FUNCTION_BLOCK "FbTON"
TITLE = 'Таймер с задержкой на включение.'

{ S7_read_back := 'true' ;
  S7_blockview := 'big'  }

AUTHOR  : VA
FAMILY  : LIB_PLC
VERSION : '2.2'

VAR_INPUT // Входные переменные, сохраняемые.
In          :BOOL := FALSE; // Вход таймера.
TimeDelayOn :DINT := 5000 ; // Время задержки включения [мс].
Ts_ms       :DINT := 100  ; // Шаг дискретизации по времени [мс].
END_VAR

VAR_OUTPUT // Выходные переменные, сохраняемые.
Out :BOOL := FALSE; // Выход таймера.
END_VAR

VAR // Внутренние переменные, сохраняемые.
Timer1 :DINT := 0; // Текущее время таймер1 [мс].
END_VAR

BEGIN

// Таймер с задержкой на включение.
//          DbTON
//    +----------------+
//    |     FbTON      |
// ->-|In           Out|->-
//   -|TimeDelayOn     |
//   -|Ts_ms           |
//    +----------------+

IF (TimeDelayOn > 0) THEN // Таймер включен.
  IF (In) THEN // На входе 1.
    IF (Out) THEN // На выходе 1.
    Out := TRUE;
    Timer1 := 0;
    ELSE // На выходе 0.
      IF (Timer1 >= TimeDelayOn) THEN // Задержка включения закончилась.
      Out := TRUE;
      Timer1 := 0;
      ELSE // Задержка включения активна.
      Out := FALSE;
      Timer1 := Timer1 + Ts_ms;
      END_IF;
    END_IF;
  ELSE // Если на входе 0 то на выходе тоже 0.
  Out := FALSE;
  Timer1 := 0;
  END_IF;
ELSE // Таймер выключен.
Out := In;
Timer1 := 0;
END_IF;

// Применение.
//
// При поступлении входного сигнала выходной сигнал появляется не сразу, а с задержкой TimeDelayOn.
// Блок может применятся как фильтр дребезга контактов дискретных входов.
// Совместно с инвертором может применяться для генерации импульсов.

// Временная характеристика.
//
//  In
//  ^
//  | TimeDelayOn           TimeDelayOn
//  |   |<--->|               |<--->|
// 1|   ***********     * *   ***********
//  |   *         *     * *   *         *
// 0*****---------*************---------*****----> t[s]
//
//  Out
//  ^
//  | TimeDelayOn           TimeDelayOn
//  |   |<--->|               |<--->|
// 1|   |     *****           |     *****
//  |   |     *   *           |     *   *
// 0***********---*******************---*****----> t[s]

// @COPYLEFT ALL WRONGS RESERVED :)
// Author: VA
// Contacts: DIY.PLC.314@gmail.com
// Date start LIB_PLC: 2014
// License: GNU GPL-2.0-or-later
// https://www.gnu.org/licenses/old-licenses/gpl-2.0.html
// https://www.youtube.com/watch?v=n1F_MfLRlX0
// https://www.youtube.com/@DIY_PLC
// https://github.com/DIYPLC/LIB_PLC
// https://oshwlab.com/diy.plc.314/PLC_HW1_SW1
// https://3dtoday.ru/3d-models/mechanical-parts/body/korpus-na-din-reiku
// https://t.me/DIY_PLC
// https://drive.google.com/drive/folders/16GDX0i07rwDrl_oPzL-lQAqMiAz3ouJV?usp=sharing

END_FUNCTION_BLOCK
